// TIA Portal V18 export
// export: Created 2026-04-18T00:00:00Z, ExportSetting WithDefaults
FUNCTION_BLOCK "FB_Comms"   // FB101, LAD
{ S7_Optimized_Access := 'TRUE' }
VERSION : 0.1
// stored: AutoNumber true, IsIECCheckEnabled false, IsRetainMemResEnabled false
BEGIN

REGION Network 1: Kiểm tra bộ đếm CTU
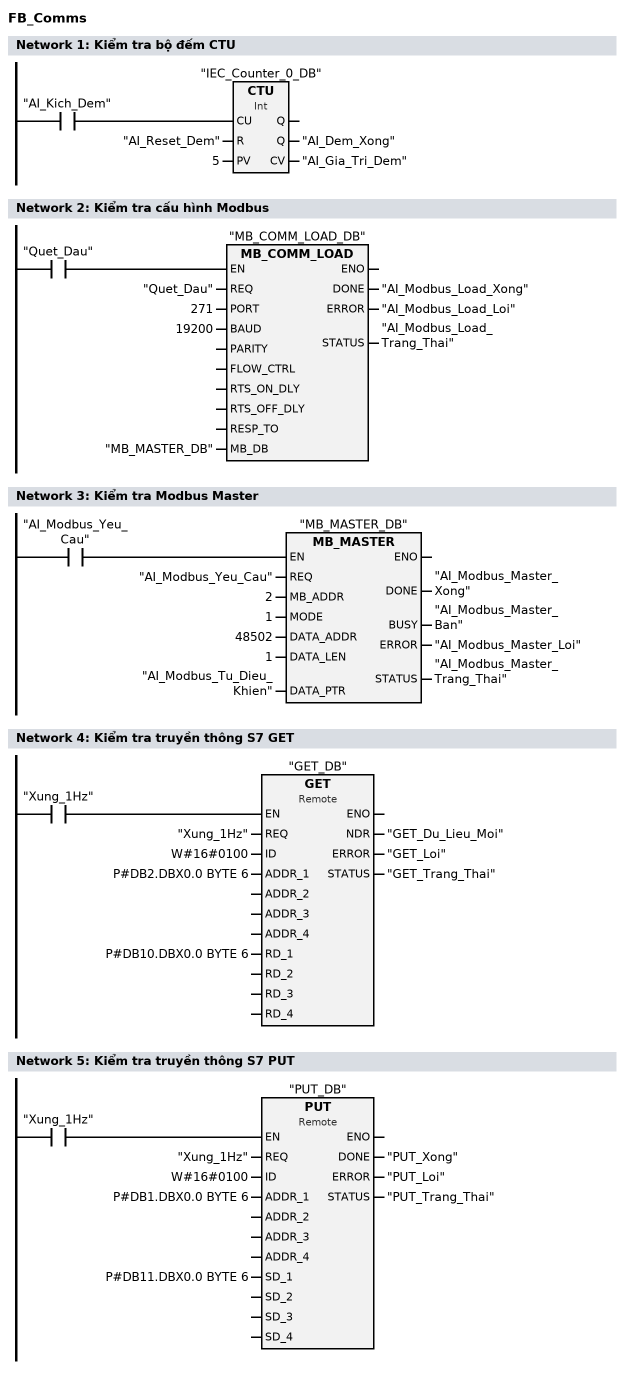
   RUNG wire#powerrail
      Contact( "AI_Kich_Dem" )
      { S7_Templates := "value_type := Int" } "IEC_Counter_0_DB".CTU(r := "AI_Reset_Dem", pv := 5, q => "AI_Dem_Xong", cv => "AI_Gia_Tri_Dem")
   END_RUNG
   // the same network as SCL:
   "IEC_Counter_0_DB".CTU(CU := "AI_Kich_Dem",
                          R := "AI_Reset_Dem",
                          PV := 5,
                          Q => "AI_Dem_Xong",
                          CV => "AI_Gia_Tri_Dem");
END_REGION

REGION Network 2: Kiểm tra cấu hình Modbus
   RUNG wire#powerrail
      Contact( "Quet_Dau" )
      "MB_COMM_LOAD_DB".MB_COMM_LOAD(REQ := "Quet_Dau", PORT := 271, BAUD := 19200, PARITY :=, FLOW_CTRL :=, RTS_ON_DLY :=, RTS_OFF_DLY :=, RESP_TO :=, MB_DB := "MB_MASTER_DB", DONE => "AI_Modbus_Load_Xong", ERROR => "AI_Modbus_Load_Loi", STATUS => "AI_Modbus_Load_Trang_Thai")
   END_RUNG
   // the same network as SCL:
   IF "Quet_Dau" THEN
       "MB_COMM_LOAD_DB"(REQ := "Quet_Dau",   // MB_COMM_LOAD
                         PORT := 271,
                         BAUD := 19200,
                         MB_DB := "MB_MASTER_DB",
                         DONE => "AI_Modbus_Load_Xong",
                         ERROR => "AI_Modbus_Load_Loi",
                         STATUS => "AI_Modbus_Load_Trang_Thai");
   END_IF;
END_REGION

REGION Network 3: Kiểm tra Modbus Master
   RUNG wire#powerrail
      Contact( "AI_Modbus_Yeu_Cau" )
      "MB_MASTER_DB".MB_MASTER(REQ := "AI_Modbus_Yeu_Cau", MB_ADDR := 2, MODE := 1, DATA_ADDR := 48502, DATA_LEN := 1, DATA_PTR := "AI_Modbus_Tu_Dieu_Khien", DONE => "AI_Modbus_Master_Xong", BUSY => "AI_Modbus_Master_Ban", ERROR => "AI_Modbus_Master_Loi", STATUS => "AI_Modbus_Master_Trang_Thai")
   END_RUNG
   // the same network as SCL:
   IF "AI_Modbus_Yeu_Cau" THEN
       "MB_MASTER_DB"(REQ := "AI_Modbus_Yeu_Cau",   // MB_MASTER
                      MB_ADDR := 2,
                      MODE := 1,
                      DATA_ADDR := 48502,
                      DATA_LEN := 1,
                      DATA_PTR := "AI_Modbus_Tu_Dieu_Khien",
                      DONE => "AI_Modbus_Master_Xong",
                      BUSY => "AI_Modbus_Master_Ban",
                      ERROR => "AI_Modbus_Master_Loi",
                      STATUS => "AI_Modbus_Master_Trang_Thai");
   END_IF;
END_REGION

REGION Network 4: Kiểm tra truyền thông S7 GET
   RUNG wire#powerrail
      Contact( "Xung_1Hz" )
      { S7_Templates := "[remote_type := Remote, local_type := Variant]" } "GET_DB".GET(REQ := "Xung_1Hz", ID := W#16#0100, ADDR_1 := P#DB2.DBX0.0 BYTE 6, ADDR_2 :=, ADDR_3 :=, ADDR_4 :=, RD_1 := P#DB10.DBX0.0 BYTE 6, RD_2 :=, RD_3 :=, RD_4 :=, NDR => "GET_Du_Lieu_Moi", ERROR => "GET_Loi", STATUS => "GET_Trang_Thai")
   END_RUNG
   // the same network as SCL:
   IF "Xung_1Hz" THEN
       "GET_DB"(REQ := "Xung_1Hz",   // GET
                ID := W#16#0100,
                ADDR_1 := P#DB2.DBX0.0 BYTE 6,
                RD_1 := P#DB10.DBX0.0 BYTE 6,
                NDR => "GET_Du_Lieu_Moi",
                ERROR => "GET_Loi",
                STATUS => "GET_Trang_Thai");
   END_IF;
END_REGION

REGION Network 5: Kiểm tra truyền thông S7 PUT
   RUNG wire#powerrail
      Contact( "Xung_1Hz" )
      { S7_Templates := "[remote_type := Remote, local_type := Variant]" } "PUT_DB".PUT(REQ := "Xung_1Hz", ID := W#16#0100, ADDR_1 := P#DB1.DBX0.0 BYTE 6, ADDR_2 :=, ADDR_3 :=, ADDR_4 :=, SD_1 := P#DB11.DBX0.0 BYTE 6, SD_2 :=, SD_3 :=, SD_4 :=, DONE => "PUT_Xong", ERROR => "PUT_Loi", STATUS => "PUT_Trang_Thai")
   END_RUNG
   // the same network as SCL:
   IF "Xung_1Hz" THEN
       "PUT_DB"(REQ := "Xung_1Hz",   // PUT
                ID := W#16#0100,
                ADDR_1 := P#DB1.DBX0.0 BYTE 6,
                SD_1 := P#DB11.DBX0.0 BYTE 6,
                DONE => "PUT_Xong",
                ERROR => "PUT_Loi",
                STATUS => "PUT_Trang_Thai");
   END_IF;
END_REGION
END_FUNCTION_BLOCK
